// TIA Portal V17 export
// export: Created 2024-06-14T09:53:03.4345504Z, ExportSetting WithDefaults, DisplayName Totally Integrated Automation Portal, DisplayVersion V17, DisplayName TIA Portal Openness, DisplayVersion V17, DisplayName TIA Portal Version Control Interface, DisplayVersion V17, DisplayName Simotion SCOUT TIA, DisplayVersion 5.4.3.0, DisplayName SINAMICS Startdrive Advanced, DisplayVersion V17 SP1 Update 1, DisplayName SINAMICS Startdrive G110M, G120, G120C, G120D, G120P, G115D, DisplayVersion V17 SP1 Update 1, DisplayName SINAMICS Startdrive G130, G150, S120, S150, SINAMICS MV, S210, DisplayVersion V17 SP1 Update 1, DisplayName STEP 7 Professional, DisplayVersion V17, DisplayName STEP 7 Safety, DisplayVersion V17, DisplayName WinCC Professional, DisplayVersion V17
DATA_BLOCK "DATA_LOG"   // DB3
{ S7_Optimized_Access := 'TRUE' }
VERSION : 0.1
// stored: AutoNumber true, DBAccessibleFromOPCUA true, IsOnlyStoredInLoadMemory false, IsRetainMemResEnabled false, IsWriteProtectedInAS false, MemoryReserve 100
   VAR
      L1_CY_ID : Int;
      L1_TARE_WT : Real;
      L1_NET_WT : Real;
      L1_GROSS_WT : Real;
      L1_CY_TYPE : Int;
      L2_CY_ID : Int;
      L2_TARE_WT : Real;
      L2_NET_WT : Real;
      L2_GROSS_WT : Real;
      L2_CY_TYPE : Int;
      MALABAR_DOMESTIC_COUNT : Int;
      MALABAR_COMMERCIAL_COUNT : Int;
      BPCL_DOMESTIC_COUNT : Int;
      BPCL_COMMERCIAL_COUNT : Int;
      TOTAL_COUNT : Int;
      L1 { S7_SetPoint := 'True'} : Array[1..6] of "uCylinderData";
      L2 { S7_SetPoint := 'True'} : Array[1..6] of "uCylinderData";
      L1_log_done { S7_SetPoint := 'True'} : Bool;
      L2_log_done : Bool;
      L1_Delet : Bool;
      L2_Delet : Bool;
      "1MINT_BIT" : Bool;
      "1M_BIT" : Bool;
      L1_TOTAL_NET_WT_CY_1 : Real;   // BPCL
      L1_TOTAL_NET_WT_CY_2 : Real;   // MALABAR
      L1_TOTAL_NET_WT_CY_3 : Real;   // BPCL
      L1_TOTAL_NET_WT_CY_4 : Real;   // MALABAR
      L2_TOTAL_NET_WT_CY_1 : Real;
      L2_TOTAL_NET_WT_CY_2 : Real;
      L2_TOTAL_NET_WT_CY_3 : Real;
      L2_TOTAL_NET_WT_CY_4 : Real;
      TOTAL_NET_WT_CY_1_D_BPCL : Real;
      TOTAL_NET_WT_CY_2_C_BPCL : Real;
      TOTAL_NET_WT_CY_3_D_MALA : Real;
      TOTAL_NET_WT_CY_4_C_MALA : Real;
   END_VAR
BEGIN
END_DATA_BLOCK
